// TIA Portal V20 export
VAR_GLOBAL   // PLC tag table "07_Energy"
   "Active energy export tariff 1(F)" AT %ID624 : Real;
   "Active energy import tariff 1(F)" AT %ID612 : Real;
   "Active power L1" AT %ID644 : Real;
   "Active power L2" AT %ID648 : Real;
   "Active power L3" AT %ID652 : Real;
   "Apparent energy tariff 1 (F)" AT %ID620 : Real;
   "Apparent power L1" AT %ID632 : Real;
   "Apparent power L2" AT %ID636 : Real;
   "Apparent power L3" AT %ID640 : Real;
   PAC3220InPut AT %I500.0 : "LER_typePAC3220Input_Status";
   "Reactive energy export tariff 1 (F)" AT %ID628 : Real;
   "Reactive energy import tariff 1 (F)" AT %ID616 : Real;
   "Reactive power L1" AT %ID656 : Real;
   "Reactive power L2" AT %ID660 : Real;
   "Reactive power L3" AT %ID664 : Real;
   PAC3220OutPut AT %Q500.0 : "LER_typePAC3220Output_Status";
END_VAR
VAR_GLOBAL CONSTANT   // user constants
   NO_OF_MACHINES : USInt := 1;   // SICAR: No of machines for EE-Monitor
   NO_OF_MEASUREPOINTS : USInt := 10;   // SICAR: No of measurepoints for EE-Monitor
   "DP_FRWA1_1_0_000CC1-KE50~DP_FRWA1_1_0_000CC1-KE50_900" : Hw_Io := 10;
END_VAR
